INTERFACE ITF_KomunikatorNadawca

END_INTERFACE

(* stored: Version 1.1.0.1
   Itf ITF_KomunikatorNadawca: Id {f2c748b8-07c6-03cf-04c2-0bcc78ff32eb} *)
